PROGRAM MAIN
VAR
END_VAR

END_PROGRAM

(* stored: Version 1.1.0.1
   POU MAIN: Id {439a731e-10f6-437d-9e9f-b6ea22b9e972} *)
